Fanuc KAREL source: compact_preamble.KL

PROGRAM NC0052
%NOLOCKGROUP
ROUTINE R
VAR
S1:INTEGER
BEGIN
S1=1
SELECT S1 OF
CASE(1):
S1=(S1 + 2)
CASE(2):
S1=(S1 + 3)
ELSE:
S1=(S1 + 1)
ENDSELECT
END R
BEGIN
R
END NC0052
